TYPE ERROR :
STRUCT
	bError : BOOL;
	nErrorCode : DINT;
END_STRUCT
END_TYPE

(* stored: Version 1.1.0.1
   DUT ERROR: Id {fb94b97b-34f6-4e50-a5c2-02d5baf5310b} *)
